VAR_GLOBAL // TIMERS
    firstRun: BOOL := TRUE;
END_VAR

(* stored: ProductVersion 3.1.0.18, Version 1.1.0.1 *)
